(* CoDeSys 2.3.9.50 project: 5D.pr6 *)
(* Libraries: STANDARD.LB6 5.6.98 12:03:02 *)

(* POU MAIN, LD *)
PROGRAM MAIN
VAR
	a: REAL := 1;
         b: REAL := -4;
	c: REAL := -45;
	b2: REAL;
	ac4: REAL;
	D: REAL;
	rootD: REAL;
	root1: REAL;
	root2: REAL;
	Calculate AT %IX0.0: BOOL;
	a1: REAL;
	a2: REAL;
END_VAR
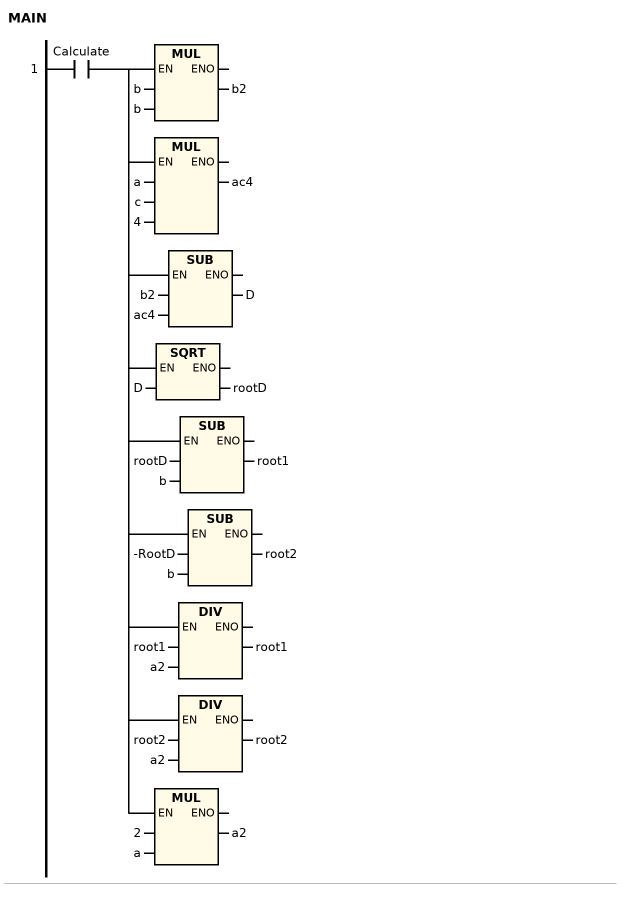
_LD_ (* Ladder Diagram *)
NETWORK 1
	[Calculate]
		EN --- MUL(b, b) => b2
		EN --- MUL(a, c, 4) => ac4
		EN --- SUB(b2, ac4) => D
		EN --- SQRT(D) => rootD
		EN --- SUB(rootD, b) => root1
		EN --- SUB(-RootD, b) => root2
		EN --- DIV(root1, a2) => root1
		EN --- DIV(root2, a2) => root2
		EN --- MUL(2, a) => a2
_END_LD_
(* the same logic as Structured Text *)
(* Network 1 *)
IF Calculate THEN
	b2 := b * b;
	ac4 := a * c * 4;
	D := b2 - ac4;
	rootD := SQRT(D);
	root1 := rootD - b;
	root2 := (-RootD) - b;
	root1 := root1 / a2;
	root2 := root2 / a2;
	a2 := 2 * a;
END_IF;
END_PROGRAM
